(* IEC 61131-3 sources: teller/JD_Teller_LC2_V11/Class/_FirstAlarm, 1 file *)

(* ---- _FirstAlarm.st ---- *)
(*!
<Class
	Name               = "_FirstAlarm"
	Revision           = "2.0"
	RealtimeTask       = "false"
	CyclicTask         = "false"
	BackgroundTask     = "false"
	Sigmatek           = "false"
	OSInterface        = "false"
	HighPriority       = "false"
	Automatic          = "false"
	UpdateMode         = "Prescan"
	SharedCommandTable = "true"
	Objectsize         = "(422,120)">
	<Channels>
		<Server Name="ActAlarmNr" Visualized="true" Initialize="false" WriteProtected="true" Retentive="false"/>
		<Server Name="AlarmTakt" Visualized="true" Initialize="false" WriteProtected="true" Retentive="false"/>
		<Client Name="SortAlgoHist" Required="true" Internal="false"/>
		<Client Name="SortAlgoTemp" Required="true" Internal="false"/>
	</Channels>
	<Network Name="_FirstAlarm">
		<!-- List of Components in this network -->
		<Components>
			<Object
				Name       = "_base"
				Class      = "_HotAlarm"
				Position   = "(218,120)"
				Visualized = "false">
				<Channels>
					<Server Name="Server0"/>
					<Client Name="Lse"/>
				</Channels>
			</Object>
		</Components>
		<Comments>
		</Comments>
		<!-- List of Connections in this network -->
		<Connections>
			<Connection Source="this.Server0" Destination="_base.Server0" Vertices="(690,210),(518,210),"/>
			<Connection Source="_base.Lse" Destination="this.Lse" Vertices="(218,210),(38,210),"/>
		</Connections>
		<!-- Headerfiles -->
		<Options>
		</Options>
	</Network>
</Class>
*)
#pragma using _HotAlarm

_FirstAlarm : CLASS
: _HotAlarm
  //Servers:
	ActAlarmNr 	: SvrCh_DINT;
	AlarmTakt 	: SvrCh_DINT;
  //Clients:
	SortAlgoTemp 	: CltCh_DINT;
	SortAlgoHist 	: CltCh_DINT;
  //Variables:
		pms 	: ^_MEM_SINGLEALARM;
		no 	: _UDWORD;
		nn 	: UDINT;
		nnn 	: UDINT;
		psa 	: ^_SINGLEALARM;
		txt 	: ^_CHAR;
		FirstTime 	: DINT;
		TimeMarkTakt 	: UDINT;
  //Functions:
				//! <Function Comment="[#ENGLISH]&#13;&#10;this method is called everytime when system wants to redraw the io&#13;&#10;&#13;&#10;pio ....... pointer to io information&#13;&#10;pr ........ pointer to result information&#13;&#10;pv ........ pointer to io variableinformation&#13;&#10;input ..... _TRUE it&apos;s an input / _FALSE it&apos;s an output&#13;&#10;&#13;&#10;for the returnstatement there are 3 different possibilities&#13;&#10;_IDLE ..... the system should goon like it is (system goes on)&#13;&#10;_IDIDIT ... i did it (system is ready)&#13;&#10;_IFAILED .. i tried to do my best, but i failed (system is ready)&#13;&#10;&#13;&#10;if you want to draw the io let&apos;s return _IDIDIT&#13;&#10;" Name="Draw"/>
	FUNCTION __CDECL VIRTUAL GLOBAL Draw
		VAR_INPUT
			pio 	: ^_IO;
			pr 	: ^_RESULT;
			pv 	: ^_VARIABLE;
			input 	: BOOL;
		END_VAR
		VAR_OUTPUT
			retcode (EAX) 	: _DOIT;
		END_VAR;
				//! <Function Comment="[#ENGLISH]&#13;&#10;this method is called everytime when system wants to get data for defined io.&#13;&#10;&#13;&#10;pr ........ pointer to result information&#13;&#10;pio ....... pointer to io information&#13;&#10;pv ........ pointer to io variableinformation&#13;&#10;input ..... _TRUE it&apos;s an input / _FALSE it&apos;s an output&#13;&#10;&#13;&#10;for the returnstatement there are 3 different possibilities&#13;&#10;_IDLE ..... the system should goon like it is (system goes on)&#13;&#10;_IDIDIT ... i did it (system is ready)&#13;&#10;_IFAILED .. i tried to do my best, but i failed (system is ready)&#13;&#10;&#13;&#10;if you want to do it let&apos;s return _IDIDIT and initialize the  structure _RESULT&#13;&#10;" Name="GetData"/>
	FUNCTION __CDECL VIRTUAL GLOBAL GetData
		VAR_INPUT
			pr 	: ^_RESULT;
			pio 	: ^_IO;
			pv 	: ^_VARIABLE;
			input 	: BOOL;
		END_VAR
		VAR_OUTPUT
			retcode (EAX) 	: _DOIT;
		END_VAR;
  //Tables:
	FUNCTION @STD
		VAR_OUTPUT
			ret_code	: CONFSTATES;
		END_VAR;
	FUNCTION GLOBAL TAB @CT_;
END_CLASS;

FUNCTION __CDECL VIRTUAL GLOBAL _FirstAlarm::Draw
	VAR_INPUT
		pio 	: ^_IO;
		pr 	: ^_RESULT;
		pv 	: ^_VARIABLE;
		input 	: BOOL;
	END_VAR
	VAR_OUTPUT
		retcode (EAX) 	: _DOIT;
	END_VAR

VAR
//  pms   : ^_MEM_SINGLEALARM;
//	psa   : ^_SINGLEALARM;
//	txt   : ^_CHAR;
	st    : BOOL;
//	no    : UDINT;
END_VAR

  if FirstTime = 0 then
    SortAlgoTemp := 2;
    SortAlgoHist := 2;
    SortAlgoTemp.Write (SortAlgoTemp);
    SortAlgoHist.Write (SortAlgoHist);
    FirstTime := 1;
  end_if;

  st  := _FALSE;
  pms := get_MEM_SINGLEALARM(_FALSE);
  no  := no_RINGBUFFER(#pms^.ringbuffer);
  nnn := 0;

  while(nnn < no) do
    nnn += 1;
    psa := pms^.ptr + rpos_RINGBUFFER(#pms^.ringbuffer, nn) * sizeof(_SINGLEALARM);
	if(psa^.state <> 0) then
      txt := create_alarmtext(psa, _FALSE, NIL);
	  if(txt <> NIL) then
	    actalarmNR := psa^.no;
      nnn := nn;  // stoppen !!
      no := nnn;
	    st := _TRUE;
      end_if;
    else
    	nn += 1;
	end_if;
  end_while;

    Graphic.Putimage(#pio^.image, DEFKOORD, DEFKOORD);
  if(st = _FALSE) then
    nn := 0; // Opnieuw als er geen alarmen meer zijn  !!
    actalarmNR := -1;
  else
    OutMultiTextAlign(txt, pio^.fillchr, #pio^.space, pio^.font, pio^.attrib, pio^.frametype, pio^.coltxt, pio^.colback, pio^.colframe, sizeof(_CHAR));
  end_if;

  retcode := _IDIDIT;

END_FUNCTION

FUNCTION __CDECL VIRTUAL GLOBAL _FirstAlarm::GetData
	VAR_INPUT
		pr 	: ^_RESULT;
		pio 	: ^_IO;
		pv 	: ^_VARIABLE;
		input 	: BOOL;
	END_VAR
	VAR_OUTPUT
		retcode (EAX) 	: _DOIT;
	END_VAR

   pms := get_MEM_SINGLEALARM(FALSE);
  pr^.ftype := RES_NUMERIC;
  pr^.rmin  := pms^.xchange;
  pr^.rmax  := pms^.xchange;
  pr^.value := pms^.xchange;
  pr^.ptr   := #pr^.value$void;

  retcode := _IDIDIT;

// #PVO  090624
  if ActAlarmNr >= 0 then
    if ops.tAbsolute - TimeMarkTakt > 500 then  // alarm signal 500ms on - - - 500ms off
      AlarmTakt := (AlarmTakt = 0);
      TimeMarkTakt := ops.tAbsolute;
    end_if;
  else
    AlarmTakt := 0;
    TimeMarkTakt := ops.tAbsolute;
  end_if;

END_FUNCTION
